(* PLC project Sin nombre, Desconocido Sin nombre 1 *)
(* stored: creationDateTime 2024-10-28T23:47:34, modificationDateTime 2024-11-01T18:42:19 *)

PROGRAM program0
  VAR
    sensor AT %IW0 : UINT;
  END_VAR
  VAR
    tope_alto : UINT := 50000;
    minimo_alto : UINT := 45000;
    minimo_superior : UINT := 50001;
    acumulador : UDINT := 0;
    acumulador0 : UDINT := 38000;
    timer : BOOL := 1;
    timer2 : BOOL := 1;
    normal : BOOL := 1;
    alto : BOOL := 0;
    superior : BOOL := 0;
    verificar : BOOL := 0;
    compara : BOOL := 0;
    divide : BOOL := 0;
  END_VAR
  VAR
    inicio AT %QX0.4 : BOOL := 0;
  END_VAR
  VAR
    timer_corrido : BOOL := 0;
    probar : BOOL := 0;
    acumular : BOOL := 0;
  END_VAR
  VAR
    luz1 AT %QX0.0 : BOOL := 0;  (* dar ubicacion *)
    luz2 AT %QX0.1 : BOOL := 0;  (* dar ubicacion *)
    pruev AT %QX0.2 : BOOL := 0;  (* 16 *)
    pruev0 AT %QX0.3 : BOOL := 0;  (* 16 *)
  END_VAR
  VAR
    TP0 : TP;
    TOF1 : TOF;
    TP3 : TP;
    CTU_LINT0 : CTU_LINT;
    TP1 : TP;
    TOF0 : TOF;
    TOF2 : TOF;
    TOF3 : TOF;
    TON2 : TON;
    TON0 : TON;
    TON1 : TON;
    TON3 : TON;
    TON4 : TON;
    TP2 : TP;
    TON5 : TON;
  END_VAR
  VAR  (* added by the conversion: wires and edge detectors of the diagram *)
    _UINT_TO_UDINT81_ENO : BOOL;
    _UINT_TO_UDINT81_OUT : UDINT;
    _ADD78_ENO : BOOL;
    _ADD78_OUT : UDINT;
    R_TRIG1 : R_TRIG;
    _UINT_TO_UDINT8_ENO : BOOL;
    _UINT_TO_UDINT8_OUT : UDINT;
    _GE93_ENO : BOOL;
    _GE93_OUT : BOOL;
    _UINT_TO_UDINT9_ENO : BOOL;
    _UINT_TO_UDINT9_OUT : UDINT;
    _LT100_ENO : BOOL;
    _LT100_OUT : BOOL;
    _UINT_TO_UDINT12_ENO : BOOL;
    _UINT_TO_UDINT12_OUT : UDINT;
    _GE104_ENO : BOOL;
    _GE104_OUT : BOOL;
    _UINT_TO_UDINT19_ENO : BOOL;
    _UINT_TO_UDINT19_OUT : UDINT;
    _LT17_ENO : BOOL;
    _LT17_OUT : BOOL;
    _GE166_ENO : BOOL;
    _GE166_OUT : BOOL;
  END_VAR

(* LD diagram, written out as Structured Text *)
probar := timer;
TP0(IN := probar AND NOT timer_corrido, PT := T#150ms);
acumular := TP0.Q;
TOF1(IN := NOT verificar AND acumular, PT := T#75ms);
timer_corrido := TOF1.Q;
TP3(IN := NOT verificar AND acumular, PT := T#10ms);
_UINT_TO_UDINT81_OUT := UINT_TO_UDINT(EN := TP3.Q, IN := sensor, ENO => _UINT_TO_UDINT81_ENO);
_ADD78_OUT := ADD(EN := TP3.Q, IN1 := acumulador, IN2 := _UINT_TO_UDINT81_OUT, ENO => _ADD78_ENO);
IF _ADD78_ENO THEN acumulador := _ADD78_OUT; END_IF;
(* normal = [3,33400,34500] 
alto = [6,34501,36800]
superior = [8,36801,38400] *)
TON4(IN := verificar, PT := T#530ms);
timer := NOT TON4.Q;
R_TRIG1(CLK := _ADD78_ENO);
TON3(IN := TP1.Q, PT := T#250ms);
CTU_LINT0(CU := R_TRIG1.Q, R := TON3.Q, PV := 7);
TP1(IN := CTU_LINT0.Q, PT := T#2s);
verificar := TP1.Q;
luz1 := NOT normal;
luz2 := NOT normal;
_UINT_TO_UDINT8_OUT := UINT_TO_UDINT(EN := TON4.Q, IN := minimo_alto, ENO => _UINT_TO_UDINT8_ENO);
_GE93_OUT := GE(EN := TON4.Q, IN1 := acumulador0, IN2 := _UINT_TO_UDINT8_OUT, ENO => _GE93_ENO);
_UINT_TO_UDINT9_OUT := UINT_TO_UDINT(EN := _GE93_OUT, IN := minimo_superior, ENO => _UINT_TO_UDINT9_ENO);
_LT100_OUT := LT(EN := _GE93_OUT, IN1 := acumulador0, IN2 := _UINT_TO_UDINT9_OUT, ENO => _LT100_ENO);
TOF2(IN := _LT100_OUT, PT := T#3280ms);
alto := TOF2.Q;
_UINT_TO_UDINT12_OUT := UINT_TO_UDINT(EN := _GE93_OUT, IN := tope_alto, ENO => _UINT_TO_UDINT12_ENO);
_GE104_OUT := GE(EN := _GE93_OUT, IN1 := acumulador0, IN2 := _UINT_TO_UDINT12_OUT, ENO => _GE104_ENO);
TOF0(IN := _GE104_OUT, PT := T#3480ms);
superior := TOF0.Q;
_UINT_TO_UDINT19_OUT := UINT_TO_UDINT(EN := TON4.Q, IN := minimo_alto, ENO => _UINT_TO_UDINT19_ENO);
_LT17_OUT := LT(EN := TON4.Q, IN1 := acumulador0, IN2 := _UINT_TO_UDINT19_OUT, ENO => _LT17_ENO);
TOF3(IN := _LT17_OUT, PT := T#3680ms);
normal := TOF3.Q;
luz1 := alto;
luz2 := superior;
TON2(IN := _LT100_OUT, PT := T#1980ms);
IF TON2.Q THEN acumulador := 0; END_IF;
TON0(IN := _GE104_OUT, PT := T#1980ms);
IF TON0.Q THEN acumulador := 0; END_IF;
TON1(IN := _LT17_OUT, PT := T#1000ms);
IF TON1.Q THEN acumulador := 0; END_IF;
_GE166_OUT := GE(EN := timer2, IN1 := sensor, IN2 := 39000, ENO => _GE166_ENO);
pruev := _GE166_OUT;
pruev0 := _ADD78_ENO;
inicio := TON4.Q;
TON5(IN := verificar, PT := T#430ms);
TP2(IN := TON5.Q, PT := T#10ms);
IF TP2.Q THEN acumulador := acumulador / 7; END_IF;
luz1 := superior;
luz2 := NOT alto;
END_PROGRAM

CONFIGURATION Config0
  RESOURCE Res0 ON PLC
    TASK task0(INTERVAL := T#20ms, PRIORITY := 0);
    PROGRAM instance0 WITH task0 : program0;
  END_RESOURCE
END_CONFIGURATION
